Staubli VAL3: User.pgx

program User()
  local num nMenu
  local pointRx pPos
begin
  userPage()
  while ()
    cls(Interfaz)
    title(Interfaz,"Pick-and-Place")
    nMenu = getKey()
    switch nmenu
      case 271
        pPos = pPointrx1[0]
      break
      case 272
        pPos = pPointrx1[1]
      break
      case 273
        pPos = pPointrx1[2]
      break
      default
        pPos=jHome
      break
    endSwitch
    if bBool2==true
      call Pick(pPos)
    else
      call Place(pPos)
    bBool2=bBool2!
  endWhile
end
